FUNCTION_BLOCK FB_ID_list_man
(* Manage a list of users ad grant access if user's tag is recognize *)

VAR_INPUT
	stUserIn	: POINTER TO stUserID;		// input ID
	stArrList : POINTER TO ARRAY [0..19] OF stUserID;
	xAdd		: BOOL;			// add a user, failed if ID is already use
	xDel		: BOOL;			// delete a user from the list, fail if ID doesn't exist
	xAccess 	: BOOL;			// modify the access level
	tRestore	: TIME;			// auto-restore time constant
	tTimeOut	: TIME;			// timeout value for the current access level. 0 is infinite
END_VAR
VAR_OUTPUT
	iCurrLevel	: enAccessLevel;	// current access level
	stLastUser	: stUserID;		// last logged user
	xFail 		: BOOL;			// last operation has failed
	xPass		: BOOL;			// access level granted or action is a success
END_VAR
VAR
	tonAutoRestore	: TON;		// Restore automatically from error
	tonTimeOut		: TON;		// Ton timeout access
	iUserIndex		: INT;		// user index from the list
END_VAR


//----------------------------------------------------------------------------------
// manage timeout
//----------------------------------------------------------------------------------
IF tTimeOut <> T#0S OR tonTimeOut.Q THEN
	tonTimeOut(IN := (NOT tonTimeOut.Q), PT := tTimeOut);
END_IF
IF tonTimeOut.Q THEN
	iCurrLevel := enAccessLevel.logged_out;
END_IF

//----------------------------------------------------------------------------------
// Restore all the error flag (in case of retry, too)
//----------------------------------------------------------------------------------
tonAutoRestore(IN := (xFail OR xPass), PT := tRestore);
IF tonAutoRestore.Q OR xAdd OR xDel OR xAccess THEN
	xFail := FALSE;
	xPass := FALSE;
END_IF

//----------------------------------------------------------------------------------
// compute input acctions 
//----------------------------------------------------------------------------------
IF xAdd THEN
	IF add_user(stArrList, stUserIn) THEN
		xPass := TRUE;
	ELSE
		xFail := TRUE;
	END_IF
END_IF

IF xDel THEN
	IF delete_user(stArrList, stUserIn) THEN
		xPass := TRUE;
	ELSE
		xFail := TRUE;
	END_IF
END_IF

IF xAccess THEN
	iUserIndex := find_user_in_list(stArrList, stUserIn);
	IF iUserIndex > 0 THEN
		stLastUser := stArrList^[iUserIndex];
		iCurrLevel := stArrList^[iUserIndex].bLevel;
		xPass := TRUE;
	ELSE
		xFail := TRUE;
	END_IF
END_IF

METHOD PRIVATE add_user : BOOL
 (* add a user to the list. Return false is the list is full *)
VAR_INPUT
	list	: POINTER TO ARRAY [0..19] OF stUserID;	// list of user
	user	: POINTER TO stUserID;					// user to add
END_VAR
VAR
	i	: INT;
	free_index	: INT;	// index of the free spot
END_VAR
add_user := FALSE;

// Monkey user checks
IF 0 = LEN(user^.sName) OR THIS^.is_tag_empty(user^.bArrTag) 
	OR (user^.bLevel < 0) OR (user^.bLevel > enAccessLevel.max_) THEN
	RETURN;
END_IF

IF THIS^.is_user_in_list(list, user) THEN
	RETURN;
END_IF

free_index := THIS^.find_free_index(list);

IF free_index < 0 THEN
	RETURN;
END_IF

list^[free_index] := user^;
add_user := TRUE;
END_METHOD

METHOD PRIVATE delete_user : BOOL
 (* delete a user to the list. Return false when the target user hasn't been found *)
VAR_INPUT
	list	: POINTER TO ARRAY [0..19] OF stUserID;	// list of user
	user	: POINTER TO stUserID;					// user to add
END_VAR
VAR
	i	: INT;
	user_index	: INT;	// index of the user to delete
END_VAR
delete_user := FALSE;

// Monkey user checks
IF THIS^.is_tag_empty(user^.bArrTag) THEN
	RETURN;
END_IF

user_index := THIS^.find_user_in_list(list, user);

IF user_index < 0 THEN
	RETURN;
END_IF

memset( ADR(list[user_index]), 0, SIZEOF(stUserID));

delete_user := TRUE;
END_METHOD

METHOD PRIVATE find_free_index : INT
(* Get the free spot of the array.
 * If none found, return value is -1
 * If a spot is found, then it return the index of the free spot
 *)
VAR_INPUT
	list	: POINTER TO ARRAY [0..19] OF stUserID;	// list of user
END_VAR
VAR
	i	: INT;
END_VAR
FOR i:=0 TO 19 BY 1 DO
	IF THIS^.is_tag_empty(list^[i].bArrTag) THEN
		find_free_index := i;
		RETURN;
	END_IF
END_FOR
find_free_index := -1;
END_METHOD

METHOD PRIVATE find_user_in_list : INT
(* Get the user location in the user list.
 * If the user is not found, the value -1 is returned
 * If the user is found, the index of the location of the user is returned
 *)
VAR_INPUT
	list	: POINTER TO ARRAY [0..19] OF stUserID;	// list of user
	user	: POINTER TO stUserID;						// user to check
END_VAR
VAR
	i	: INT;
END_VAR
FOR i:=0 TO 19 BY 1 DO
	IF THIS^.is_tag_equal(list^[i].bArrTag, user^.bArrTag) THEN
		find_user_in_list := i;
		RETURN;
	END_IF
END_FOR
find_user_in_list := -1;
END_METHOD

METHOD PRIVATE is_tag_empty : BOOL
(* Return TRUE if all the fields from a tag is emtpy *)
VAR_INPUT
	tag		: ARRAY [0..7] OF BYTE;	// input tag
END_VAR
VAR
	i	: INT;
END_VAR
is_tag_empty := FALSE;
FOR i:=0 TO 7 BY 1 DO
	IF 0 <> tag[i] THEN
		RETURN;
	END_IF
END_FOR
is_tag_empty := TRUE;
END_METHOD

METHOD PRIVATE is_tag_equal : BOOL
(* compare 2 tags. Return TRUE when the 2 tags matches *)
VAR_INPUT
	tag1	: ARRAY [0..7] OF BYTE;		// First tag to compare
	tag2	: ARRAY [0..7] OF BYTE;		// Second tag to compare
END_VAR
VAR
	i	: INT;
END_VAR
is_tag_equal := FALSE;
FOR i:=0 TO 7 BY 1 DO
	IF 0 <> MEMCMP(ADR(tag1), ADR(tag2), 8) THEN
		RETURN;
	END_IF
END_FOR
is_tag_equal := TRUE;
END_METHOD

METHOD PRIVATE is_user_in_list : BOOL
(* Return TRUE when the given user is in the given list *)
VAR_INPUT
	list	: POINTER TO ARRAY [0..19] OF stUserID;	// list of user
	user	: POINTER TO stUserID;						// user to check
END_VAR
VAR
	i	: INT;
END_VAR
is_user_in_list := FALSE;
FOR i:=0 TO 19 BY 1 DO
	IF THIS^.is_tag_equal(list^[i].bArrTag, user^.bArrTag) THEN
		is_user_in_list := TRUE;
	END_IF
END_FOR
END_METHOD

END_FUNCTION_BLOCK

(* stored: Version 1.1.0.1, ProductVersion 3.1.4024.6
   POU FB_ID_list_man: Id {9b76b178-bc7a-4898-96bb-151fb9de157f}, SpecialFunc None
   Method add_user: Id {ec6f172b-ecea-40d8-b7c8-1a4c94a13711}
   Method delete_user: Id {2087d1e1-27c3-4e59-b568-6c624f23de81}
   Method find_free_index: Id {ecedf067-ce69-4f3c-bac5-2f5747b5224a}
   Method find_user_in_list: Id {4a6d07f3-e447-4e9f-82ad-8a9e4bf3686c}
   Method is_tag_empty: Id {c9145936-ac3c-42d2-9e07-1221c6a18460}
   Method is_tag_equal: Id {6e668225-facf-40fe-9bec-e158a886dcfe}
   Method is_user_in_list: Id {b5f39436-ed7d-406d-9c23-2ba3190a11f0} *)
